{attribute 'pack_mode' := '1'}
TYPE ST_PLCMsg:
STRUCT
    version: DINT; (* Version of set of PLC<->CCS messages. *)
END_STRUCT
END_TYPE

(* stored: Version 1.1.0.1, ProductVersion 3.1.4022.18
   DUT ST_PLCMsg: Id {ac8f3146-7045-4105-9ae0-2b0a3953c3f3} *)
